# B&R Automation Studio project RTFProj (part 5)

#### test.c - Init, cyclic, exit code
```c
/*********************************************************************************************
* B&R Automation - Perfection in Automation (https://www.br-automation.com)
    ******************************************************************************************
    * Program 	    : Master's Thesis - Soccer Table (Table Football - real game)
    * Author  	    : Roman Parak
    * Created 	    : date ...
	* University    : Brno University of Technology(BUT)
	* Faculty       : Faculty of Mechanical Engineering(FME)
	* Study Program : Applied Computer Science and Control
	* Institute     : Institute of Automation and Computer Science
**********************************************************************************************
* Implementation OF PROGRAM Test(Real_Game/Technology/Test/Program/test.h)
**********************************************************************************************/

/*************************** LIBRARIES *********************************/
#include <bur/plc.h>
#include <bur/plctypes.h>
#include <stdio.h>
#include <math.h>

#include "rp_funcx1.h"
#include "Structures/test_str.h"
#include "Functions/test_fce.h"

#ifdef _DEFAULT_INCLUDES
	#include <AsDefault.h>
#endif

/*************************** DEFINITIONS *******************************/
#define EACH_FORMATION 1;

/************************ LOCAL VARIABLES ******************************/
// struct - MpAlarmX
_LOCAL MpAlarmXListUIConnectType AlarmListUI_ConnectType;
_LOCAL MpAlarmXHistoryUIConnectType AlarmHistoryUI_ConnectType;
// udint
_LOCAL UDINT alarm_device_address;
// bool
_LOCAL BOOL start;
_LOCAL BOOL stop;
// usint
_LOCAL USINT max_numberOfFormation;
_LOCAL USINT i_axisNum;
// lreal
_LOCAL LREAL temp_lin;
_LOCAL LREAL temp_rot;
_LOCAL LREAL define_posRotary;
_LOCAL LREAL angle_ofRotation;
// state machine
_LOCAL rp_MainSteps soccer_step;

/**********************************************************************************************************/
/********************************************** INIT PROGRAM **********************************************/
/**********************************************************************************************************/
void _INIT ProgramInit(void)
{
    /*********************************** Declaration variables **********************************/
    // generally
    max_numberOfFormation = EACH_FORMATION;

    // axis type -> MAPP -> Name Mapp axes for testing
    // linear
    //gLinkAxes_linear[0] = gk_mappAxisL;
    /*
    gLinkAxes_linear[1] = df_mappAxisL;
    gLinkAxes_linear[2] = md_mappAxisL;
    gLinkAxes_linear[3] = fw_mappAxisL;
    */
    // rotary
    //gLinkAxes_rotary[0] = gk_mappAxisR;
   	/*
    gLinkAxes_rotary[1] = df_mappAxisR;
    gLinkAxes_rotary[2] = md_mappAxisR;
    gLinkAxes_rotary[3] = fw_mappAxisR;
    */
    /************************************ Control of AlarmX ************************************/

    // adjustment device name
    alarm_device_address = (UDINT) strcpy(mp_alarmX.deviceName_no1_exp,"EXPORT_HISTORY");
    // MpAlarmX Core
    mp_alarmX.mp_core.MpLink         = &gAlarmXCore;
    mp_alarmX.mp_core.Enable         = 1;
    // MpAlarmX ListUI
    mp_alarmX.mp_listUI.MpLink       = &gAlarmXCore;
    mp_alarmX.mp_listUI.Enable       = 1;
    mp_alarmX.mp_listUI.UIConnect    = &AlarmListUI_ConnectType;
    // MpAlarmX History
    mp_alarmX.mp_history.MpLink      = &gAlarmXHistory;
    mp_alarmX.mp_history.Enable      = 1;
    mp_alarmX.mp_history.DeviceName  = &mp_alarmX.deviceName_no1_exp;
    // MpAlarmX HistoryUI
    mp_alarmX.mp_historyUI.MpLink    = &gAlarmXHistory;
    mp_alarmX.mp_historyUI.Enable    = 1;
    mp_alarmX.mp_historyUI.UIConnect = &AlarmHistoryUI_ConnectType;

    /************************************* Control of Axes **************************************/

    for(i_axisNum = 0; i_axisNum <= max_numberOfFormation - 1; i_axisNum++){
        // initialization ACOPOS variables through function(get_axisParam), that returns two variables type of UDINT
        // into the structure -> axesAcopos(have two parameters : linear, rotary)
        axis_acopos = get_axisParam(i_axisNum);
        // linear -> LinMot
        // linear axis basic
        mp_Axis.mp_axisLinear[i_axisNum].Enable     = 1;
        mp_Axis.mp_axisLinear[i_axisNum].MpLink     = &gLinkAxes_linear[i_axisNum];
        mp_Axis.mp_axisLinear[i_axisNum].Parameters = &mp_Axis.param_axisLinear[i_axisNum];
        mp_Axis.mp_axisLinear[i_axisNum].Axis       = axis_acopos.linear;
		// initialization parameters -> linear
		mp_Axis.param_axisLinear[i_axisNum].Home.Mode 	 		 	     = mpAXIS_HOME_MODE_BLOCK_TORQUE;
		mp_Axis.param_axisLinear[i_axisNum].Home.Position 		  	     = 900;
		mp_Axis.param_axisLinear[i_axisNum].Home.StartVelocity   		 = 350;
		mp_Axis.param_axisLinear[i_axisNum].Home.HomingVelocity  		 = 450;
		mp_Axis.param_axisLinear[i_axisNum].Home.Acceleration    		 = 350;
		mp_Axis.param_axisLinear[i_axisNum].Home.StartDirection  		 = mpAXIS_HOME_DIR_POSITIVE;
		mp_Axis.param_axisLinear[i_axisNum].Home.HomingDirection 		 = mpAXIS_HOME_DIR_NEGATIVE;
		mp_Axis.param_axisLinear[i_axisNum].Home.TorqueLimit	 		 = 0.05;
		mp_Axis.param_axisLinear[i_axisNum].Home.PositionErrorStopLimit	 = 900;
        // linear cyclic set
        mp_Axis.mp_cyclicSetLinear[i_axisNum].Enable     = 1;
        mp_Axis.mp_cyclicSetLinear[i_axisNum].MpLink     = &gLinkAxes_linear[i_axisNum];
        mp_Axis.mp_cyclicSetLinear[i_axisNum].Parameters = &mp_Axis.param_cyclicSetLinear[i_axisNum];
		// config
		mp_Axis.mp_configAxisLinear[i_axisNum].Enable 		 = 1;
		mp_Axis.mp_configAxisLinear[i_axisNum].MpLink 		 = &gLinkAxes_linear[i_axisNum];
		mp_Axis.mp_configAxisLinear[i_axisNum].Configuration = &mp_Axis.param_configAxisLinear[i_axisNum];
        // rotary -> EnDat
        // rotary axis basic
        mp_Axis.mp_axisRotary[i_axisNum].Enable     = 1;
        mp_Axis.mp_axisRotary[i_axisNum].MpLink     = &gLinkAxes_rotary[i_axisNum];
        mp_Axis.mp_axisRotary[i_axisNum].Parameters = &mp_Axis.param_axisRotary[i_axisNum];
        mp_Axis.mp_axisRotary[i_axisNum].Axis       = axis_acopos.rotary;
        // rotary cyclic set
        mp_Axis.mp_cyclicSetRotary[i_axisNum].Enable     = 1;
        mp_Axis.mp_cyclicSetRotary[i_axisNum].MpLink     = &gLinkAxes_rotary[i_axisNum];
        mp_Axis.mp_cyclicSetRotary[i_axisNum].Parameters = &mp_Axis.param_cyclicSetRotary[i_axisNum];
		// config
		mp_Axis.mp_configAxisRotary[i_axisNum].Enable 		 = 1;
		mp_Axis.mp_configAxisRotary[i_axisNum].MpLink 		 = &gLinkAxes_rotary[i_axisNum];
		mp_Axis.mp_configAxisRotary[i_axisNum].Configuration = &mp_Axis.param_configAxisRotary[i_axisNum];
		// temperature - linear
		mp_Axis.param_axisLinear[i_axisNum].CyclicRead.MotorTempMode = mpAXIS_READ_POLLING_1s;
		// temperature - rotary
		mp_Axis.param_axisRotary[i_axisNum].CyclicRead.MotorTempMode = mpAXIS_READ_POLLING_1s;
    }
	// initializatiom temp
	temp_lin = 0;
	temp_rot = 0;
	define_posRotary = 118520697;
	angle_ofRotation = 0;
	// initialization state machine
	soccer_step = STEP_INITIALIZATION;
}

/**********************************************************************************************************/
/********************************************** MAIN PROGRAM **********************************************/
/**********************************************************************************************************/
void _CYCLIC ProgramCyclic(void)
{
	// initializatiom temp
	temp_lin = mp_Axis.mp_axisLinear[0].Info.CyclicRead.MotorTemperature.Value;
	temp_rot = mp_Axis.mp_axisRotary[0].Info.CyclicRead.MotorTemperature.Value;

	switch(soccer_step)
	{
		case STEP_INITIALIZATION:
			{
				if(mp_Axis.mp_axisLinear[0].Active == 1 && mp_Axis.mp_axisRotary[0].Active == 1){
					angle_ofRotation = get_rotationalPostition(mp_Axis.mp_axisRotary[0].Position,define_posRotary);

					if(labs(angle_ofRotation) <= 3600){
						mp_Axis.param_axisRotary[0].Home.Position = angle_ofRotation;
						soccer_step = STEP_INITIALIZATION0;
					}
				}
			}
			break;
		case STEP_INITIALIZATION0:
			{
				if(mp_Axis.mp_axisLinear[0].Error == 1 && mp_Axis.mp_axisRotary[0].Error == 0){
					soccer_step = STEP_ERROR1;
				}else if(mp_Axis.mp_axisLinear[0].StatusID < 0 || mp_Axis.mp_axisRotary[0].StatusID < 0){
					soccer_step = STEP_ERROR2;
				}else {
					if(mp_Axis.mp_axisLinear[0].IsHomed == 1 && mp_Axis.mp_axisRotary[0].IsHomed == 1){
						soccer_step = STEP_RUN7;
					}else{
						soccer_step = STEP_INITIALIZATION1;
					}
				}
			}
			break;
		case STEP_INITIALIZATION1:
			{
				if(start == 1){
					mp_Axis.mp_axisLinear[0].Power = 1;
					mp_Axis.mp_axisRotary[0].Power = 1;

					if(mp_alarmX.mp_core.ActiveAlarms == 1){
						soccer_step = STEP_ERROR1;
					}else if(stop == 1){
						soccer_step = STEP_STOP1;
					}else{
						if(mp_Axis.mp_axisLinear[0].PowerOn == 1 && mp_Axis.mp_axisRotary[0].PowerOn == 1){
							soccer_step = STEP_INITIALIZATION2;
						}
					}
				}
			}
			break;
		case STEP_INITIALIZATION2:
			{
				mp_Axis.mp_axisLinear[0].Update = 1;
				mp_Axis.mp_axisRotary[0].Update = 1;

				if(mp_alarmX.mp_core.ActiveAlarms == 1){
					soccer_step = STEP_ERROR1;
				}else if(stop == 1){
					soccer_step = STEP_STOP1;
				}else{
					if(mp_Axis.mp_axisLinear[0].UpdateDone == 1 && mp_Axis.mp_axisRotary[0].UpdateDone == 1){
						mp_Axis.mp_axisLinear[0].Update = 0;
						mp_Axis.mp_axisRotary[0].Update = 0;
						soccer_step = STEP_INITIALIZATION3;
					}
				}
			}
			break;
		case STEP_INITIALIZATION3:
			{
				mp_Axis.mp_axisRotary[0].Home = 1;

				if(mp_alarmX.mp_core.ActiveAlarms == 1){
					soccer_step = STEP_ERROR1;
				}else if(stop == 1){
					soccer_step = STEP_STOP1;
				}else{
					if(mp_Axis.mp_axisRotary[0].IsHomed == 1){
						mp_Axis.mp_axisRotary[0].Home = 0;
						soccer_step = STEP_INITIALIZATION4;
					}
				}
			}
			break;
		case STEP_INITIALIZATION4:
			{
				mp_Axis.param_cyclicSetRotary[0].Acceleration = 2000;
				mp_Axis.param_cyclicSetRotary[0].Deceleration = 2000;
				mp_Axis.param_cyclicSetRotary[0].PositionModeMaxVelocity = 85000;
				mp_Axis.mp_cyclicSetRotary[0].Velocity 	 = 1000;
				mp_Axis.mp_cyclicSetRotary[0].Position	 = 0;

				mp_Axis.mp_cyclicSetRotary[0].Update = 1;
				if(mp_alarmX.mp_core.ActiveAlarms == 1){
					soccer_step = STEP_ERROR1;
				}else if(stop == 1){
					soccer_step = STEP_STOP1;
				}else{
					if(mp_Axis.mp_cyclicSetRotary[0].UpdateDone == 1){
						mp_Axis.mp_cyclicSetRotary[0].Update = 0;
						if(mp_Axis.mp_cyclicSetRotary[0].CommandBusy == 0 && mp_Axis.mp_cyclicSetRotary[0].CyclicSetActive == 0){
							soccer_step = STEP_INITIALIZATION5;
						}
					}
				}
			}
			break;
		case STEP_INITIALIZATION5:
			{
				mp_Axis.mp_cyclicSetRotary[0].CyclicPosition = 1;
				if(mp_alarmX.mp_core.ActiveAlarms == 1){
					soccer_step = STEP_ERROR1;
				}else if(stop == 1){
					soccer_step = STEP_STOP1;
				}else{
					if(mp_Axis.mp_cyclicSetRotary[0].Info.SlavePosition == 0){
						mp_Axis.mp_cyclicSetRotary[0].CyclicPosition = 0;
						if(mp_Axis.mp_cyclicSetRotary[0].CommandBusy == 0 && mp_Axis.mp_cyclicSetRotary[0].CyclicSetActive == 0){
							soccer_step = STEP_INITIALIZATION6;
						}
					}
				}
			}
			break;
		case STEP_INITIALIZATION6:
			{
				mp_Axis.mp_axisLinear[0].Home = 1;

				if(mp_alarmX.mp_core.ActiveAlarms == 1){
					soccer_step = STEP_ERROR1;
				}else if(stop == 1){
					soccer_step = STEP_STOP1;
				}else{
					if(mp_Axis.mp_axisLinear[0].IsHomed == 1){
						mp_Axis.mp_axisLinear[0].Home = 0;
						soccer_step = STEP_START;
					}
				}
			}
			break;
		case STEP_START:
			{
				mp_Axis.param_cyclicSetLinear[0].Acceleration = 400000;
				mp_Axis.param_cyclicSetLinear[0].Deceleration = 400000;
				mp_Axis.param_cyclicSetLinear[0].PositionModeMaxVelocity = 30000;
				mp_Axis.mp_cyclicSetLinear[0].Velocity = 19000;
				mp_Axis.mp_cyclicSetLinear[0].Position = 0;

				mp_Axis.mp_cyclicSetLinear[0].Update = 1;
				if(mp_alarmX.mp_core.ActiveAlarms == 1){
					soccer_step = STEP_ERROR1;
				}else if(stop == 1){
					soccer_step = STEP_STOP1;
				}else{
					if(mp_Axis.mp_cyclicSetLinear[0].UpdateDone == 1){
						mp_Axis.mp_cyclicSetLinear[0].Update = 0;
						if(mp_Axis.mp_cyclicSetLinear[0].CommandBusy == 0 && mp_Axis.mp_cyclicSetLinear[0].CyclicSetActive == 0){
							soccer_step = STEP_RUN1;
						}
					}
				}
			}
			break;
		case STEP_RUN1:
			{
				mp_Axis.mp_cyclicSetLinear[0].CyclicPosition = 1;
				if(mp_alarmX.mp_core.ActiveAlarms == 1){
					soccer_step = STEP_ERROR1;
				}else if(stop == 1){
					soccer_step = STEP_STOP1;
				}else{
					if(mp_Axis.mp_cyclicSetLinear[0].Info.SlavePosition == 0){
						mp_Axis.mp_cyclicSetLinear[0].CyclicPosition = 0;
						if(mp_Axis.mp_cyclicSetLinear[0].CommandBusy == 0 && mp_Axis.mp_cyclicSetLinear[0].CyclicSetActive == 0){
							soccer_step = STEP_RUN2;
						}
					}
				}
			}
			break;
		case STEP_RUN2:
			{
				mp_Axis.param_cyclicSetRotary[0].Acceleration = 125000;
				mp_Axis.param_cyclicSetRotary[0].Deceleration = 125000;
				mp_Axis.param_cyclicSetRotary[0].PositionModeMaxVelocity = 85000;
				mp_Axis.mp_cyclicSetRotary[0].Velocity 	 = 10000;
				mp_Axis.mp_cyclicSetRotary[0].Position	 = -800;

				mp_Axis.mp_cyclicSetRotary[0].Update = 1;
				if(mp_alarmX.mp_core.ActiveAlarms == 1){
					soccer_step = STEP_ERROR1;
				}else if(stop == 1){
					soccer_step = STEP_STOP1;
				}else{
					if(mp_Axis.mp_cyclicSetRotary[0].UpdateDone == 1){
						mp_Axis.mp_cyclicSetRotary[0].Update = 0;
						if(mp_Axis.mp_cyclicSetRotary[0].CommandBusy == 0 && mp_Axis.mp_cyclicSetRotary[0].CyclicSetActive == 0){
							soccer_step = STEP_RUN3;
						}
					}
				}
			}
			break;
		case STEP_RUN3:
			{
				mp_Axis.mp_cyclicSetRotary[0].CyclicPosition = 1;
				if(mp_alarmX.mp_core.ActiveAlarms == 1){
					soccer_step = STEP_ERROR1;
				}else if(stop == 1){
					soccer_step = STEP_STOP1;
				}else{
					if(mp_Axis.mp_cyclicSetRotary[0].Info.SlavePosition == -800){
						mp_Axis.mp_cyclicSetRotary[0].CyclicPosition = 0;
						if(mp_Axis.mp_cyclicSetRotary[0].CommandBusy == 0 && mp_Axis.mp_cyclicSetRotary[0].CyclicSetActive == 0){
							soccer_step = STEP_RUN4;
						}
					}
				}
			}
			break;
		case STEP_RUN4:
			{
				mp_Axis.param_cyclicSetRotary[0].Acceleration = 125000;
				mp_Axis.param_cyclicSetRotary[0].Deceleration = 125000;
				mp_Axis.param_cyclicSetRotary[0].PositionModeMaxVelocity = 85000;
				mp_Axis.mp_cyclicSetRotary[0].Velocity 	 = 10000;
				mp_Axis.mp_cyclicSetRotary[0].Position	 = 800;

				mp_Axis.mp_cyclicSetRotary[0].Update = 1;
				if(mp_alarmX.mp_core.ActiveAlarms == 1){
					soccer_step = STEP_ERROR1;
				}else if(stop == 1){
					soccer_step = STEP_STOP1;
				}else{
					if(mp_Axis.mp_cyclicSetRotary[0].UpdateDone == 1){
						mp_Axis.mp_cyclicSetRotary[0].Update = 0;
						if(mp_Axis.mp_cyclicSetRotary[0].CommandBusy == 0 && mp_Axis.mp_cyclicSetRotary[0].CyclicSetActive == 0){
							soccer_step = STEP_RUN5;
						}
					}
				}
			}
			break;
		case STEP_RUN5:
			{
				mp_Axis.mp_cyclicSetRotary[0].CyclicPosition = 1;
				if(mp_alarmX.mp_core.ActiveAlarms == 1){
					soccer_step = STEP_ERROR1;
				}else if(stop == 1){
					soccer_step = STEP_STOP1;
				}else{
					if(mp_Axis.mp_cyclicSetRotary[0].Info.SlavePosition == 800){
						mp_Axis.mp_cyclicSetRotary[0].CyclicPosition = 0;
						if(mp_Axis.mp_cyclicSetRotary[0].CommandBusy == 0 && mp_Axis.mp_cyclicSetRotary[0].CyclicSetActive == 0){
							soccer_step = STEP_RUN6;
						}
					}
				}
			}
			break;
		case STEP_RUN6:
			{
				/*======================= END HOME =======================*/
				mp_Axis.param_cyclicSetRotary[0].Acceleration = 125000;
				mp_Axis.param_cyclicSetRotary[0].Deceleration = 125000;
				mp_Axis.param_cyclicSetRotary[0].PositionModeMaxVelocity = 85000;
				mp_Axis.mp_cyclicSetRotary[0].Velocity 	 = 10000;
				mp_Axis.mp_cyclicSetRotary[0].Position	 = 0;

				mp_Axis.mp_cyclicSetRotary[0].Update = 1;
				if(mp_alarmX.mp_core.ActiveAlarms == 1){
					soccer_step = STEP_ERROR1;
				}else if(stop == 1){
					soccer_step = STEP_STOP1;
				}else{
					if(mp_Axis.mp_cyclicSetRotary[0].UpdateDone == 1){
						mp_Axis.mp_cyclicSetRotary[0].Update = 0;
						if(mp_Axis.mp_cyclicSetRotary[0].CommandBusy == 0 && mp_Axis.mp_cyclicSetRotary[0].CyclicSetActive == 0){
							soccer_step = STEP_RUN7;
						}
					}
				}
			}
			break;
		case STEP_RUN7:
			{
				/*======================= START CYCLE =======================*/
				mp_Axis.mp_cyclicSetRotary[0].CyclicPosition = 1;
				if(mp_alarmX.mp_core.ActiveAlarms == 1){
					soccer_step = STEP_ERROR1;
				}else if(stop == 1){
					soccer_step = STEP_STOP1;
				}else{
					if(mp_Axis.mp_cyclicSetRotary[0].Info.SlavePosition == 0){
						mp_Axis.mp_cyclicSetRotary[0].CyclicPosition = 0;
						if(mp_Axis.mp_cyclicSetRotary[0].CommandBusy == 0 && mp_Axis.mp_cyclicSetRotary[0].CyclicSetActive == 0){
							soccer_step = STEP_RUN8;
						}
					}
				}
			}
			break;
		case STEP_RUN8:
			{
				// 250000,20000
				mp_Axis.param_cyclicSetLinear[0].Acceleration = 125000;
				mp_Axis.param_cyclicSetLinear[0].Deceleration = 125000;
				mp_Axis.param_cyclicSetLinear[0].PositionModeMaxVelocity = 30000;
				mp_Axis.mp_cyclicSetLinear[0].Velocity = 10000;
				mp_Axis.mp_cyclicSetLinear[0].Position = -800;

				mp_Axis.mp_cyclicSetLinear[0].Update = 1;
				if(mp_alarmX.mp_core.ActiveAlarms == 1){
					soccer_step = STEP_ERROR1;
				}else if(stop == 1){
					soccer_step = STEP_STOP1;
				}else{
					if(mp_Axis.mp_cyclicSetLinear[0].UpdateDone == 1){
						mp_Axis.mp_cyclicSetLinear[0].Update = 0;
						if(mp_Axis.mp_cyclicSetLinear[0].CommandBusy == 0 && mp_Axis.mp_cyclicSetLinear[0].CyclicSetActive == 0){
							soccer_step = STEP_RUN9;
						}
					}
				}
			}
			break;
		case STEP_RUN9:
			{
				mp_Axis.mp_cyclicSetLinear[0].CyclicPosition = 1;
				if(mp_alarmX.mp_core.ActiveAlarms == 1){
					soccer_step = STEP_ERROR1;
				}else if(stop == 1){
					soccer_step = STEP_STOP1;
				}else{
					if(mp_Axis.mp_cyclicSetLinear[0].Info.SlavePosition == -800){
						mp_Axis.mp_cyclicSetLinear[0].CyclicPosition = 0;
						if(mp_Axis.mp_cyclicSetLinear[0].CommandBusy == 0 && mp_Axis.mp_cyclicSetLinear[0].CyclicSetActive == 0){
							soccer_step = STEP_RUN10; // STEP_RUN24
						}
					}
				}
			}
			break;
		case STEP_RUN10:
			{
				mp_Axis.param_cyclicSetRotary[0].Acceleration = 31250;
				mp_Axis.param_cyclicSetRotary[0].Deceleration = 31250;
				mp_Axis.param_cyclicSetRotary[0].PositionModeMaxVelocity = 85000;
				mp_Axis.mp_cyclicSetRotary[0].Velocity 	 = 5000;
				mp_Axis.mp_cyclicSetRotary[0].Position	 = -800;

				mp_Axis.mp_cyclicSetRotary[0].Update = 1;
				if(mp_alarmX.mp_core.ActiveAlarms == 1){
					soccer_step = STEP_ERROR1;
				}else if(stop == 1){
					soccer_step = STEP_STOP1;
				}else{
					if(mp_Axis.mp_cyclicSetRotary[0].UpdateDone == 1){
						mp_Axis.mp_cyclicSetRotary[0].Update = 0;
						if(mp_Axis.mp_cyclicSetRotary[0].CommandBusy == 0 && mp_Axis.mp_cyclicSetRotary[0].CyclicSetActive == 0){
							soccer_step = STEP_RUN11;
						}
					}
				}
			}
			break;
		case STEP_RUN11:
			{
				mp_Axis.mp_cyclicSetRotary[0].CyclicPosition = 1;
				if(mp_alarmX.mp_core.ActiveAlarms == 1){
					soccer_step = STEP_ERROR1;
				}else if(stop == 1){
					soccer_step = STEP_STOP1;
				}else{
					if(mp_Axis.mp_cyclicSetRotary[0].Info.SlavePosition == -800){
						mp_Axis.mp_cyclicSetRotary[0].CyclicPosition = 0;
						if(mp_Axis.mp_cyclicSetRotary[0].CommandBusy == 0 && mp_Axis.mp_cyclicSetRotary[0].CyclicSetActive == 0){
							soccer_step = STEP_RUN12;
						}
					}
				}
			}
			break;
		case STEP_RUN12:
			{
				mp_Axis.param_cyclicSetRotary[0].Acceleration = 31250;
				mp_Axis.param_cyclicSetRotary[0].Deceleration = 31250;
				mp_Axis.param_cyclicSetRotary[0].PositionModeMaxVelocity = 85000;
				mp_Axis.mp_cyclicSetRotary[0].Velocity 	 = 5000;
				mp_Axis.mp_cyclicSetRotary[0].Position	 = 800;

				mp_Axis.mp_cyclicSetRotary[0].Update = 1;
				if(mp_alarmX.mp_core.ActiveAlarms == 1){
					soccer_step = STEP_ERROR1;
				}else if(stop == 1){
					soccer_step = STEP_STOP1;
				}else{
					if(mp_Axis.mp_cyclicSetRotary[0].UpdateDone == 1){
						mp_Axis.mp_cyclicSetRotary[0].Update = 0;
						if(mp_Axis.mp_cyclicSetRotary[0].CommandBusy == 0 && mp_Axis.mp_cyclicSetRotary[0].CyclicSetActive == 0){
							soccer_step = STEP_RUN13;
						}
					}
				}
			}
			break;
		case STEP_RUN13:
			{
				mp_Axis.mp_cyclicSetRotary[0].CyclicPosition = 1;
				if(mp_alarmX.mp_core.ActiveAlarms == 1){
					soccer_step = STEP_ERROR1;
				}else if(stop == 1){
					soccer_step = STEP_STOP1;
				}else{
					if(mp_Axis.mp_cyclicSetRotary[0].Info.SlavePosition == 800){
						mp_Axis.mp_cyclicSetRotary[0].CyclicPosition = 0;
						if(mp_Axis.mp_cyclicSetRotary[0].CommandBusy == 0 && mp_Axis.mp_cyclicSetRotary[0].CyclicSetActive == 0){
							soccer_step = STEP_RUN14;
						}
					}
				}
			}
			break;
		case STEP_RUN14:
			{
				mp_Axis.param_cyclicSetRotary[0].Acceleration = 31250;
				mp_Axis.param_cyclicSetRotary[0].Deceleration = 31250;
				mp_Axis.param_cyclicSetRotary[0].PositionModeMaxVelocity = 85000;
				mp_Axis.mp_cyclicSetRotary[0].Velocity 	 = 5000;
				mp_Axis.mp_cyclicSetRotary[0].Position	 = 0;

				mp_Axis.mp_cyclicSetRotary[0].Update = 1;
				if(mp_alarmX.mp_core.ActiveAlarms == 1){
					soccer_step = STEP_ERROR1;
				}else if(stop == 1){
					soccer_step = STEP_STOP1;
				}else{
					if(mp_Axis.mp_cyclicSetRotary[0].UpdateDone == 1){
						mp_Axis.mp_cyclicSetRotary[0].Update = 0;
						if(mp_Axis.mp_cyclicSetRotary[0].CommandBusy == 0 && mp_Axis.mp_cyclicSetRotary[0].CyclicSetActive == 0){
							soccer_step = STEP_RUN15;
						}
					}
				}
			}
			break;
		case STEP_RUN15:
			{
				mp_Axis.mp_cyclicSetRotary[0].CyclicPosition = 1;
				if(mp_alarmX.mp_core.ActiveAlarms == 1){
					soccer_step = STEP_ERROR1;
				}else if(stop == 1){
					soccer_step = STEP_STOP1;
				}else{
					if(mp_Axis.mp_cyclicSetRotary[0].Info.SlavePosition == 0){
						mp_Axis.mp_cyclicSetRotary[0].CyclicPosition = 0;
						if(mp_Axis.mp_cyclicSetRotary[0].CommandBusy == 0 && mp_Axis.mp_cyclicSetRotary[0].CyclicSetActive == 0){
							soccer_step = STEP_RUN16; // STEP_RUN24
						}
					}
				}
			}
			break;
		case STEP_RUN16:
			{
				mp_Axis.param_cyclicSetLinear[0].Acceleration = 600;
				mp_Axis.param_cyclicSetLinear[0].Deceleration = 600;
				mp_Axis.param_cyclicSetLinear[0].PositionModeMaxVelocity = 30000;
				mp_Axis.mp_cyclicSetLinear[0].Velocity = 2500;
				mp_Axis.mp_cyclicSetLinear[0].Position = 0;

				mp_Axis.mp_cyclicSetLinear[0].Update = 1;
				if(mp_alarmX.mp_core.ActiveAlarms == 1){
					soccer_step = STEP_ERROR1;
				}else if(stop == 1){
					soccer_step = STEP_STOP1;
				}else{
					if(mp_Axis.mp_cyclicSetLinear[0].UpdateDone == 1){
						mp_Axis.mp_cyclicSetLinear[0].Update = 0;
						if(mp_Axis.mp_cyclicSetLinear[0].CommandBusy == 0 && mp_Axis.mp_cyclicSetLinear[0].CyclicSetActive == 0){
							soccer_step = STEP_RUN17;
						}
					}
				}
			}
			break;
		case STEP_RUN17:
			{
				mp_Axis.mp_cyclicSetLinear[0].CyclicPosition = 1;
				if(mp_alarmX.mp_core.ActiveAlarms == 1){
					soccer_step = STEP_ERROR1;
				}else if(stop == 1){
					soccer_step = STEP_STOP1;
				}else{
					if(mp_Axis.mp_cyclicSetLinear[0].Info.SlavePosition == 0){
						mp_Axis.mp_cyclicSetLinear[0].CyclicPosition = 0;
						if(mp_Axis.mp_cyclicSetLinear[0].CommandBusy == 0 && mp_Axis.mp_cyclicSetLinear[0].CyclicSetActive == 0){
							soccer_step = STEP_RUN18;
						}
					}
				}
			}
			break;
		case STEP_RUN18:
			{
				mp_Axis.param_cyclicSetRotary[0].Acceleration = 3900000;
				mp_Axis.param_cyclicSetRotary[0].Deceleration = 3900000;
				mp_Axis.param_cyclicSetRotary[0].PositionModeMaxVelocity = 85000;
				mp_Axis.mp_cyclicSetRotary[0].Velocity 	 = 84000;
				mp_Axis.mp_cyclicSetRotary[0].Position	 = -800;

				mp_Axis.mp_cyclicSetRotary[0].Update = 1;
				if(mp_alarmX.mp_core.ActiveAlarms == 1){
					soccer_step = STEP_ERROR1;
				}else if(stop == 1){
					soccer_step = STEP_STOP1;
				}else{
					if(mp_Axis.mp_cyclicSetRotary[0].UpdateDone == 1){
						mp_Axis.mp_cyclicSetRotary[0].Update = 0;
						if(mp_Axis.mp_cyclicSetRotary[0].CommandBusy == 0 && mp_Axis.mp_cyclicSetRotary[0].CyclicSetActive == 0){
							soccer_step = STEP_RUN19;
						}
					}
				}
			}
			break;
		case STEP_RUN19:
			{
				mp_Axis.mp_cyclicSetRotary[0].CyclicPosition = 1;
				if(mp_alarmX.mp_core.ActiveAlarms == 1){
					soccer_step = STEP_ERROR1;
				}else if(stop == 1){
					soccer_step = STEP_STOP1;
				}else{
					if(mp_Axis.mp_cyclicSetRotary[0].Info.SlavePosition == -800){
						mp_Axis.mp_cyclicSetRotary[0].CyclicPosition = 0;
						if(mp_Axis.mp_cyclicSetRotary[0].CommandBusy == 0 && mp_Axis.mp_cyclicSetRotary[0].CyclicSetActive == 0){
							soccer_step = STEP_RUN20;
						}
					}
				}
			}
			break;
		case STEP_RUN20:
			{
				mp_Axis.param_cyclicSetRotary[0].Acceleration = 3900000;
				mp_Axis.param_cyclicSetRotary[0].Deceleration = 3900000;
				mp_Axis.param_cyclicSetRotary[0].PositionModeMaxVelocity = 85000;
				mp_Axis.mp_cyclicSetRotary[0].Velocity 	 = 80000;
				mp_Axis.mp_cyclicSetRotary[0].Position	 = 800;

				mp_Axis.mp_cyclicSetRotary[0].Update = 1;
				if(mp_alarmX.mp_core.ActiveAlarms == 1){
					soccer_step = STEP_ERROR1;
				}else if(stop == 1){
					soccer_step = STEP_STOP1;
				}else{
					if(mp_Axis.mp_cyclicSetRotary[0].UpdateDone == 1){
						mp_Axis.mp_cyclicSetRotary[0].Update = 0;
						if(mp_Axis.mp_cyclicSetRotary[0].CommandBusy == 0 && mp_Axis.mp_cyclicSetRotary[0].CyclicSetActive == 0){
							soccer_step = STEP_RUN21;
						}
					}
				}
			}
			break;
		case STEP_RUN21:
			{
				mp_Axis.mp_cyclicSetRotary[0].CyclicPosition = 1;
				if(mp_alarmX.mp_core.ActiveAlarms == 1){
					soccer_step = STEP_ERROR1;
				}else if(stop == 1){
					soccer_step = STEP_STOP1;
				}else{
					if(mp_Axis.mp_cyclicSetRotary[0].Info.SlavePosition == 800){
						mp_Axis.mp_cyclicSetRotary[0].CyclicPosition = 0;
						if(mp_Axis.mp_cyclicSetRotary[0].CommandBusy == 0 && mp_Axis.mp_cyclicSetRotary[0].CyclicSetActive == 0){
							soccer_step = STEP_RUN22;
						}
					}
				}
			}
			break;
		case STEP_RUN22:
			{
				mp_Axis.param_cyclicSetRotary[0].Acceleration = 3900000;
				mp_Axis.param_cyclicSetRotary[0].Deceleration = 3900000;
				mp_Axis.param_cyclicSetRotary[0].PositionModeMaxVelocity = 85000;
				mp_Axis.mp_cyclicSetRotary[0].Velocity 	 = 80000;
				mp_Axis.mp_cyclicSetRotary[0].Position	 = 0;

				mp_Axis.mp_cyclicSetRotary[0].Update = 1;
				if(mp_alarmX.mp_core.ActiveAlarms == 1){
					soccer_step = STEP_ERROR1;
				}else if(stop == 1){
					soccer_step = STEP_STOP1;
				}else{
					if(mp_Axis.mp_cyclicSetRotary[0].UpdateDone == 1){
						mp_Axis.mp_cyclicSetRotary[0].Update = 0;
						if(mp_Axis.mp_cyclicSetRotary[0].CommandBusy == 0 && mp_Axis.mp_cyclicSetRotary[0].CyclicSetActive == 0){
							soccer_step = STEP_RUN23;
						}
					}
				}
			}
			break;
		case STEP_RUN23:
			{
				mp_Axis.mp_cyclicSetRotary[0].CyclicPosition = 1;
				if(mp_alarmX.mp_core.ActiveAlarms == 1){
					soccer_step = STEP_ERROR1;
				}else if(stop == 1){
					soccer_step = STEP_STOP1;
				}else{
					if(mp_Axis.mp_cyclicSetRotary[0].Info.SlavePosition == 0){
						mp_Axis.mp_cyclicSetRotary[0].CyclicPosition = 0;
						if(mp_Axis.mp_cyclicSetRotary[0].CommandBusy == 0 && mp_Axis.mp_cyclicSetRotary[0].CyclicSetActive == 0){
							soccer_step = STEP_RUN24;
						}
					}
				}
			}
			break;
		case STEP_RUN24:
			{
				// 250000, 20000
				mp_Axis.param_cyclicSetLinear[0].Acceleration = 281250;
				mp_Axis.param_cyclicSetLinear[0].Deceleration = 281250;
				mp_Axis.param_cyclicSetLinear[0].PositionModeMaxVelocity = 30000;
				mp_Axis.mp_cyclicSetLinear[0].Velocity = 15000;
				mp_Axis.mp_cyclicSetLinear[0].Position = 800;

				mp_Axis.mp_cyclicSetLinear[0].Update = 1;
				if(mp_alarmX.mp_core.ActiveAlarms == 1){
					soccer_step = STEP_ERROR1;
				}else if(stop == 1){
					soccer_step = STEP_STOP1;
				}else{
					if(mp_Axis.mp_cyclicSetLinear[0].UpdateDone == 1){
						mp_Axis.mp_cyclicSetLinear[0].Update = 0;
						if(mp_Axis.mp_cyclicSetLinear[0].CommandBusy == 0 && mp_Axis.mp_cyclicSetLinear[0].CyclicSetActive == 0){
							soccer_step = STEP_RUN25;
						}
					}
				}
			}
			break;
		case STEP_RUN25:
			{
				mp_Axis.mp_cyclicSetLinear[0].CyclicPosition = 1;
				if(mp_alarmX.mp_core.ActiveAlarms == 1){
					soccer_step = STEP_ERROR1;
				}else if(stop == 1){
					soccer_step = STEP_STOP1;
				}else{
					if(mp_Axis.mp_cyclicSetLinear[0].Info.SlavePosition == 800){
						mp_Axis.mp_cyclicSetLinear[0].CyclicPosition = 0;
						if(mp_Axis.mp_cyclicSetLinear[0].CommandBusy == 0 && mp_Axis.mp_cyclicSetLinear[0].CyclicSetActive == 0){
							soccer_step = STEP_RUN26; // STEP_RUN8
						}
					}
				}
			}
			break;
		case STEP_RUN26:
			{
				mp_Axis.param_cyclicSetRotary[0].Acceleration = 3125000;
				mp_Axis.param_cyclicSetRotary[0].Deceleration = 3125000;
				mp_Axis.param_cyclicSetRotary[0].PositionModeMaxVelocity = 85000;
				mp_Axis.mp_cyclicSetRotary[0].Velocity 	 = 50000;
				mp_Axis.mp_cyclicSetRotary[0].Position	 = -800;

				mp_Axis.mp_cyclicSetRotary[0].Update = 1;
				if(mp_alarmX.mp_core.ActiveAlarms == 1){
					soccer_step = STEP_ERROR1;
				}else if(stop == 1){
					soccer_step = STEP_STOP1;
				}else{
					if(mp_Axis.mp_cyclicSetRotary[0].UpdateDone == 1){
						mp_Axis.mp_cyclicSetRotary[0].Update = 0;
						if(mp_Axis.mp_cyclicSetRotary[0].CommandBusy == 0 && mp_Axis.mp_cyclicSetRotary[0].CyclicSetActive == 0){
							soccer_step = STEP_RUN27;
						}
					}
				}
			}
			break;
		case STEP_RUN27:
			{
				mp_Axis.mp_cyclicSetRotary[0].CyclicPosition = 1;
				if(mp_alarmX.mp_core.ActiveAlarms == 1){
					soccer_step = STEP_ERROR1;
				}else if(stop == 1){
					soccer_step = STEP_STOP1;
				}else{
					if(mp_Axis.mp_cyclicSetRotary[0].Info.SlavePosition == -800){
						mp_Axis.mp_cyclicSetRotary[0].CyclicPosition = 0;
						if(mp_Axis.mp_cyclicSetRotary[0].CommandBusy == 0 && mp_Axis.mp_cyclicSetRotary[0].CyclicSetActive == 0){
							soccer_step = STEP_RUN28;
						}
					}
				}
			}
			break;
		case STEP_RUN28:
			{
				mp_Axis.param_cyclicSetRotary[0].Acceleration = 11300;
				mp_Axis.param_cyclicSetRotary[0].Deceleration = 11300;
				mp_Axis.param_cyclicSetRotary[0].PositionModeMaxVelocity = 85000;
				mp_Axis.mp_cyclicSetRotary[0].Velocity 	 = 3000;
				mp_Axis.mp_cyclicSetRotary[0].Position	 = 800;

				mp_Axis.mp_cyclicSetRotary[0].Update = 1;
				if(mp_alarmX.mp_core.ActiveAlarms == 1){
					soccer_step = STEP_ERROR1;
				}else if(stop == 1){
					soccer_step = STEP_STOP1;
				}else{
					if(mp_Axis.mp_cyclicSetRotary[0].UpdateDone == 1){
						mp_Axis.mp_cyclicSetRotary[0].Update = 0;
						if(mp_Axis.mp_cyclicSetRotary[0].CommandBusy == 0 && mp_Axis.mp_cyclicSetRotary[0].CyclicSetActive == 0){
							soccer_step = STEP_RUN29;
						}
					}
				}
			}
			break;
		case STEP_RUN29:
			{
				mp_Axis.mp_cyclicSetRotary[0].CyclicPosition = 1;
				if(mp_alarmX.mp_core.ActiveAlarms == 1){
					soccer_step = STEP_ERROR1;
				}else if(stop == 1){
					soccer_step = STEP_STOP1;
				}else{
					if(mp_Axis.mp_cyclicSetRotary[0].Info.SlavePosition == 800){
						mp_Axis.mp_cyclicSetRotary[0].CyclicPosition = 0;
						if(mp_Axis.mp_cyclicSetRotary[0].CommandBusy == 0 && mp_Axis.mp_cyclicSetRotary[0].CyclicSetActive == 0){
							soccer_step = STEP_RUN30;
						}
					}
				}
			}
			break;
		case STEP_RUN30:
			{
				mp_Axis.param_cyclicSetRotary[0].Acceleration = 1000;
				mp_Axis.param_cyclicSetRotary[0].Deceleration = 1000;
				mp_Axis.param_cyclicSetRotary[0].PositionModeMaxVelocity = 85000;
				mp_Axis.mp_cyclicSetRotary[0].Velocity 	 = 1000;
				mp_Axis.mp_cyclicSetRotary[0].Position	 = 0;

				mp_Axis.mp_cyclicSetRotary[0].Update = 1;
				if(mp_alarmX.mp_core.ActiveAlarms == 1){
					soccer_step = STEP_ERROR1;
				}else if(stop == 1){
					soccer_step = STEP_STOP1;
				}else{
					if(mp_Axis.mp_cyclicSetRotary[0].UpdateDone == 1){
						mp_Axis.mp_cyclicSetRotary[0].Update = 0;
						if(mp_Axis.mp_cyclicSetRotary[0].CommandBusy == 0 && mp_Axis.mp_cyclicSetRotary[0].CyclicSetActive == 0){
							soccer_step = STEP_RUN31;
						}
					}
				}
			}
			break;
		case STEP_RUN31:
			{
				mp_Axis.mp_cyclicSetRotary[0].CyclicPosition = 1;
				if(mp_alarmX.mp_core.ActiveAlarms == 1){
					soccer_step = STEP_ERROR1;
				}else if(stop == 1){
					soccer_step = STEP_STOP1;
				}else{
					if(mp_Axis.mp_cyclicSetRotary[0].Info.SlavePosition == 0){
						mp_Axis.mp_cyclicSetRotary[0].CyclicPosition = 0;
						if(mp_Axis.mp_cyclicSetRotary[0].CommandBusy == 0 && mp_Axis.mp_cyclicSetRotary[0].CyclicSetActive == 0){
							soccer_step = STEP_RUN32; //STEP_RUN8
						}
					}
				}
			}
			break;
		case STEP_RUN32:
			{
				mp_Axis.param_cyclicSetLinear[0].Acceleration = 440000;
				mp_Axis.param_cyclicSetLinear[0].Deceleration = 440000;
				mp_Axis.param_cyclicSetLinear[0].PositionModeMaxVelocity = 30000;
				mp_Axis.mp_cyclicSetLinear[0].Velocity = 20000;
				mp_Axis.mp_cyclicSetLinear[0].Position = 0;

				mp_Axis.mp_cyclicSetLinear[0].Update = 1;
				if(mp_alarmX.mp_core.ActiveAlarms == 1){
					soccer_step = STEP_ERROR1;
				}else if(stop == 1){
					soccer_step = STEP_STOP1;
				}else{
					if(mp_Axis.mp_cyclicSetLinear[0].UpdateDone == 1){
						mp_Axis.mp_cyclicSetLinear[0].Update = 0;
						if(mp_Axis.mp_cyclicSetLinear[0].CommandBusy == 0 && mp_Axis.mp_cyclicSetLinear[0].CyclicSetActive == 0){
							soccer_step = STEP_RUN33;
						}
					}
				}
			}
			break;
		case STEP_RUN33:
			{
				mp_Axis.mp_cyclicSetLinear[0].CyclicPosition = 1;
				if(mp_alarmX.mp_core.ActiveAlarms == 1){
					soccer_step = STEP_ERROR1;
				}else if(stop == 1){
					soccer_step = STEP_STOP1;
				}else{
					if(mp_Axis.mp_cyclicSetLinear[0].Info.SlavePosition == 0){
						mp_Axis.mp_cyclicSetLinear[0].CyclicPosition = 0;
						if(mp_Axis.mp_cyclicSetLinear[0].CommandBusy == 0 && mp_Axis.mp_cyclicSetLinear[0].CyclicSetActive == 0){
							soccer_step = STEP_RUN34;
						}
					}
				}
			}
			break;
		case STEP_RUN34:
			{
				mp_Axis.param_cyclicSetRotary[0].Acceleration = 3900000;
				mp_Axis.param_cyclicSetRotary[0].Deceleration = 3900000;
				mp_Axis.param_cyclicSetRotary[0].PositionModeMaxVelocity = 85000;
				mp_Axis.mp_cyclicSetRotary[0].Velocity 	 = 84000;
				mp_Axis.mp_cyclicSetRotary[0].Position	 = -800;

				mp_Axis.mp_cyclicSetRotary[0].Update = 1;
				if(mp_alarmX.mp_core.ActiveAlarms == 1){
					soccer_step = STEP_ERROR1;
				}else if(stop == 1){
					soccer_step = STEP_STOP1;
				}else{
					if(mp_Axis.mp_cyclicSetRotary[0].UpdateDone == 1){
						mp_Axis.mp_cyclicSetRotary[0].Update = 0;
						if(mp_Axis.mp_cyclicSetRotary[0].CommandBusy == 0 && mp_Axis.mp_cyclicSetRotary[0].CyclicSetActive == 0){
							soccer_step = STEP_RUN35;
						}
					}
				}
			}
			break;
		case STEP_RUN35:
			{
				mp_Axis.mp_cyclicSetRotary[0].CyclicPosition = 1;
				if(mp_alarmX.mp_core.ActiveAlarms == 1){
					soccer_step = STEP_ERROR1;
				}else if(stop == 1){
					soccer_step = STEP_STOP1;
				}else{
					if(mp_Axis.mp_cyclicSetRotary[0].Info.SlavePosition == -800){
						mp_Axis.mp_cyclicSetRotary[0].CyclicPosition = 0;
						if(mp_Axis.mp_cyclicSetRotary[0].CommandBusy == 0 && mp_Axis.mp_cyclicSetRotary[0].CyclicSetActive == 0){
							soccer_step = STEP_RUN36;
						}
					}
				}
			}
			break;
		case STEP_RUN36:
			{
				mp_Axis.param_cyclicSetRotary[0].Acceleration = 3900000;
				mp_Axis.param_cyclicSetRotary[0].Deceleration = 3900000;
				mp_Axis.param_cyclicSetRotary[0].PositionModeMaxVelocity = 85000;
				mp_Axis.mp_cyclicSetRotary[0].Velocity 	 = 84000;
				mp_Axis.mp_cyclicSetRotary[0].Position	 = 800;

				mp_Axis.mp_cyclicSetRotary[0].Update = 1;
				if(mp_alarmX.mp_core.ActiveAlarms == 1){
					soccer_step = STEP_ERROR1;
				}else if(stop == 1){
					soccer_step = STEP_STOP1;
				}else{
					if(mp_Axis.mp_cyclicSetRotary[0].UpdateDone == 1){
						mp_Axis.mp_cyclicSetRotary[0].Update = 0;
						if(mp_Axis.mp_cyclicSetRotary[0].CommandBusy == 0 && mp_Axis.mp_cyclicSetRotary[0].CyclicSetActive == 0){
							soccer_step = STEP_RUN37;
						}
					}
				}
			}
			break;
		case STEP_RUN37:
			{
				mp_Axis.mp_cyclicSetRotary[0].CyclicPosition = 1;
				if(mp_alarmX.mp_core.ActiveAlarms == 1){
					soccer_step = STEP_ERROR1;
				}else if(stop == 1){
					soccer_step = STEP_STOP1;
				}else{
					if(mp_Axis.mp_cyclicSetRotary[0].Info.SlavePosition == 800){
						mp_Axis.mp_cyclicSetRotary[0].CyclicPosition = 0;
						if(mp_Axis.mp_cyclicSetRotary[0].CommandBusy == 0 && mp_Axis.mp_cyclicSetRotary[0].CyclicSetActive == 0){
							soccer_step = STEP_RUN38;
						}
					}
				}
			}
			break;
		case STEP_RUN38:
			{
				mp_Axis.param_cyclicSetRotary[0].Acceleration = 61300;
				mp_Axis.param_cyclicSetRotary[0].Deceleration = 61300;
				mp_Axis.param_cyclicSetRotary[0].PositionModeMaxVelocity = 85000;
				mp_Axis.mp_cyclicSetRotary[0].Velocity 	 = 7000;
				mp_Axis.mp_cyclicSetRotary[0].Position	 = 0;

				mp_Axis.mp_cyclicSetRotary[0].Update = 1;
				if(mp_alarmX.mp_core.ActiveAlarms == 1){
					soccer_step = STEP_ERROR1;
				}else if(stop == 1){
					soccer_step = STEP_STOP1;
				}else{
					if(mp_Axis.mp_cyclicSetRotary[0].UpdateDone == 1){
						mp_Axis.mp_cyclicSetRotary[0].Update = 0;
						if(mp_Axis.mp_cyclicSetRotary[0].CommandBusy == 0 && mp_Axis.mp_cyclicSetRotary[0].CyclicSetActive == 0){
							soccer_step = STEP_RUN39;
						}
					}
				}
			}
			break;
		case STEP_RUN39:
			{
				mp_Axis.mp_cyclicSetRotary[0].CyclicPosition = 1;
				if(mp_alarmX.mp_core.ActiveAlarms == 1){
					soccer_step = STEP_ERROR1;
				}else if(stop == 1){
					soccer_step = STEP_STOP1;
				}else{
					if(mp_Axis.mp_cyclicSetRotary[0].Info.SlavePosition == 0){
						mp_Axis.mp_cyclicSetRotary[0].CyclicPosition = 0;
						if(mp_Axis.mp_cyclicSetRotary[0].CommandBusy == 0 && mp_Axis.mp_cyclicSetRotary[0].CyclicSetActive == 0){
							soccer_step = STEP_RUN8;
						}
					}
				}
			}
			break;
		case STEP_RUN40:
			{
				if(mp_alarmX.mp_core.ActiveAlarms == 1){
					soccer_step = STEP_ERROR1;
				}else if(stop == 1){
					soccer_step = STEP_STOP1;
				}else{
				}
			}
			break;
		case STEP_STOP1:
			{
				start = 0;
				mp_Axis.mp_axisLinear[0].Stop = 1;
				mp_Axis.mp_axisRotary[0].Stop = 1;

				if(mp_alarmX.mp_core.ActiveAlarms == 1){
					soccer_step = STEP_ERROR1;
				}else if(stop == 0){
					mp_Axis.mp_axisLinear[0].Stop = 0;
					mp_Axis.mp_axisRotary[0].Stop = 0;
					soccer_step = STEP_INITIALIZATION0;
				}
			}
			break;
		case STEP_ERROR1:
			{
				start = 0;
				stop  = 0;
				mp_Axis.mp_axisLinear[0].Stop = 0;
				mp_Axis.mp_axisRotary[0].Stop = 0;
				mp_Axis.mp_axisLinear[0].Power = 0;
				mp_Axis.mp_axisRotary[0].Power = 0;

				mp_Axis.mp_axisLinear[0].ErrorReset = 1;
				mp_Axis.mp_axisRotary[0].ErrorReset = 1;

				if(mp_Axis.mp_axisLinear[0].Error == 0 && mp_Axis.mp_axisRotary[0].Error == 0){
					mp_Axis.mp_axisLinear[0].ErrorReset = 0;
					mp_Axis.mp_axisRotary[0].ErrorReset = 0;

					soccer_step = STEP_INITIALIZATION0;
				}

			}
			break;
		case STEP_ERROR2:
			{
				mp_Axis.mp_axisLinear[0].ErrorReset = 1;
				mp_Axis.mp_axisRotary[0].ErrorReset = 1;

				if(mp_Axis.mp_axisLinear[0].StatusID >= 0 && mp_Axis.mp_axisRotary[0].StatusID >= 0){
					mp_Axis.mp_axisLinear[0].ErrorReset = 0;
					mp_Axis.mp_axisRotary[0].ErrorReset = 0;

					soccer_step = STEP_INITIALIZATION0;
				}
			}
			break;
	}

    /************************** Call function & function blocks **************************/
    // AlarmX
    MpAlarmXCore(&mp_alarmX.mp_core);
    MpAlarmXListUI(&mp_alarmX.mp_listUI);
    MpAlarmXHistory(&mp_alarmX.mp_history);
    MpAlarmXHistoryUI(&mp_alarmX.mp_historyUI);
    // Active AxisBasic & AxisCyclicSet -> through the individual functions
    start_axesBasic(max_numberOfFormation,&mp_Axis.mp_axisLinear,&mp_Axis.mp_axisRotary);
    start_axesCyclic(max_numberOfFormation,&mp_Axis.mp_cyclicSetLinear,&mp_Axis.mp_cyclicSetRotary);

}
```

#### test_str.h
```c
/*********************************************************************************************
* B&R Automation - Perfection in Automation (https://www.br-automation.com)
    ******************************************************************************************
    * Program 	    : Master's Thesis - Soccer Table (Table Football - real game)
    * Author  	    : Roman Parak
    * Created 	    : date ...
	* University    : Brno University of Technology(BUT)
	* Faculty       : Faculty of Mechanical Engineering(FME)
	* Study Program : Applied Computer Science and Control
	* Institute     : Institute of Automation and Computer Science
**********************************************************************************************
* Implementation OF PROGRAM Test(Real_Game/Technolog/Test/Structures/test_str.h)
**********************************************************************************************/

/*************************** LIBRARIES *********************************/
#include <bur/plc.h>
#include <bur/plctypes.h>
#include <AsString.h>
#include <AsWStr.h>

#ifdef _DEFAULT_INCLUDES
    #include <AsDefault.h>
#endif

/**********************************************************************************************************/
/************************************** STRUCTURE TYPE ****************************************************/
/**********************************************************************************************************/

/***************************** ALARM ***********************************/
typedef struct mappAlarmX_STR{
    // list
    struct MpAlarmXCore   mp_core;
    struct MpAlarmXListUI mp_listUI;
    // history
    struct    MpAlarmXHistory mp_history;
    struct    MpAlarmXHistoryUI mp_historyUI;
    plcstring deviceName_no1_exp[21];
} mappAlarmX_STR;

/***************************** AXIS ************************************/
typedef struct mappAxisBasic_STR{
    // === Linear Axes === //
    // axis basic
    struct MpAxisBasic        mp_axisLinear[4];
    struct MpAxisBasicParType param_axisLinear[4];
    // cyclic set
    struct MpAxisCyclicSet        mp_cyclicSetLinear[4];
    struct MpAxisCyclicSetParType param_cyclicSetLinear[4];
	// config
	struct MpAxisBasicConfig mp_configAxisLinear[4];
	struct MpAxisBasicConfigType param_configAxisLinear[4];
    // === Rotary Axes === //
    // axis basic
    struct MpAxisBasic        mp_axisRotary[4];
    struct MpAxisBasicParType param_axisRotary[4];
    // cyclic set
    struct MpAxisCyclicSet        mp_cyclicSetRotary[4];
    struct MpAxisCyclicSetParType param_cyclicSetRotary[4];
	// config
	struct MpAxisBasicConfig mp_configAxisRotary[4];
	struct MpAxisBasicConfigType param_configAxisRotary[4];
} mappAxisBasic_STR;

// auxiliary structures
typedef struct axesAcopos{
    UDINT linear;
    UDINT rotary;
}axesAcopos;

/**********************************************************************************************************/
/**************************************** GLOBAL VARIABLES ************************************************/
/**********************************************************************************************************/
// my structures
_GLOBAL mappAlarmX_STR mp_alarmX;
_GLOBAL mappAxisBasic_STR mp_Axis;
_GLOBAL axesAcopos axis_acopos;

// axis type -> ACOPOS
// goalkeeper
_GLOBAL ACP10AXIS_typ gkLinearW;
_GLOBAL ACP10AXIS_typ gkRotaryW;
// defender
/*
_GLOBAL ACP10AXIS_typ dfLinearX;
_GLOBAL ACP10AXIS_typ dfRotaryX;
// midfielder
_GLOBAL ACP10AXIS_typ mdLinearY;
_GLOBAL ACP10AXIS_typ mdRotaryY;
// forward
_GLOBAL ACP10AXIS_typ fwLinearZ;
_GLOBAL ACP10AXIS_typ fwRotaryZ;
*/
// axis type -> MAPP
_GLOBAL struct MpComIdentType gLinkAxes_rotary[4];
_GLOBAL struct MpComIdentType gLinkAxes_linear[4];

/**********************************************************************************************************/
/************************************** FUNCTIONS & FUNCTIONS BLOCKS **************************************/
/**********************************************************************************************************/
void start_axesBasic(USINT num_ofAxes,struct MpAxisBasic* axis_linear,struct MpAxisBasic* axis_rotary);
void start_axesCyclic(USINT num_ofAxes,struct MpAxisCyclicSet* cyclic_linear,struct MpAxisCyclicSet* cyclic_rotary);
struct axesAcopos get_axisParam(int idx_ofIteration);
```

#### test_fce.h
```c
/*********************************************************************************************
* B&R Automation - Perfection in Automation (https://www.br-automation.com)
    ******************************************************************************************
    * Program 	    : Master's Thesis - Soccer Table (Table Football - real game)
    * Author  	    : Roman Parak
    * Created 	    : date ...
	* University    : Brno University of Technology(BUT)
	* Faculty       : Faculty of Mechanical Engineering(FME)
	* Study Program : Applied Computer Science and Control
	* Institute     : Institute of Automation and Computer Science
**********************************************************************************************
* Implementation OF PROGRAM Test(Real_Game/Technolog/table_football/Functions/test_mapp_fce.h)
**********************************************************************************************/

/*************************** LIBRARIES *********************************/
#include <bur/plc.h>
#include <bur/plctypes.h>
#include <AsString.h>
#include <standard.h>
#include <AsWStr.h>
#include <stdio.h>
#include <math.h>

#ifdef _DEFAULT_INCLUDES
    #include <AsDefault.h>
#endif

/**********************************************************************************************************/
/************************************** FUNCTIONS & FUNCTIONS BLOCKS **************************************/
/**********************************************************************************************************/
void start_axesBasic(USINT num_ofAxes,struct MpAxisBasic* axis_linear,struct MpAxisBasic* axis_rotary){
    int i;
    // Axis Basic
    // function to start the individual axes
    // the cycle is carried out through number of axes
    for(i = 0; i <= num_ofAxes - 1; i++){
        // mapp axis basic
        MpAxisBasic(&axis_linear[i]);
        MpAxisBasic(&axis_rotary[i]);
    }
}

void start_axesCyclic(USINT num_ofAxes,struct MpAxisCyclicSet* cyclic_linear,struct MpAxisCyclicSet* cyclic_rotary){
    int i;
    // Axis Cyclic Set
    // function to start the individual axes
    // the cycle is carried out through number of axes
    for(i = 0; i <= num_ofAxes - 1; i++){
        // mapp axis cyclic set
        MpAxisCyclicSet(&cyclic_linear[i]);
        MpAxisCyclicSet(&cyclic_rotary[i]);
    }
}

struct axesAcopos get_axisParam(int idx_ofIteration){
    // input into the function is number of iteration(in the init part)
    // create auxiliary structures and enumeration type(for state machine)
    struct axesAcopos a;
    typedef enum {aNUM1 = 0, aNUM2, aNUM3, aNUM4}wState_ofAxes;
    wState_ofAxes new_idx; // initialize state machine
    new_idx = idx_ofIteration;
    // gradually into the state machine loading indexes from initialization part
    // and this run the function blocks
    // each state of machine has initialization both engines linear and rotary, on its own axis
    // output of this function is structure, that has two parameters(linear,rotary axis)
    switch(new_idx){
        case aNUM1:
			// Name real axes
			/*
            // goalkeeper
            a.linear = &gkLinearW;
            a.rotary = &gkRotaryW;
            return a;
            break;
        case aNUM2:
            // defender
            a.linear = &dfLinearX;
            a.rotary = &dfRotaryX;
            return a;
            break;
        case aNUM3:
            // midfielder
            a.linear = &mdLinearY;
            a.rotary = &mdRotaryY;
            return a;
            break;
        case aNUM4:
            // forward
            a.linear = &fwLinearZ;
            a.rotary = &fwRotaryZ;
            break;
        */
    }
}
```

### Program Logical/Real_Game/Technology/cam_sens_sd_s (ANSIC) - Lubo,Radek program for real game.

#### main_real.c - Init, cyclic, exit code
```c
/*********************************************************************************************
* B&R Automation - Perfection in Automation (https://www.br-automation.com)
    ******************************************************************************************
    * Program 	    : Bachelor's Thesis
    * Author  	    : Lubomir Bubenik, Radek Otradovský
    * Created 	    : date ...
	* University    : Brno University of Technology(BUT)
	* Faculty       : Faculty of Mechanical Engineering(FME), Faculty of Electrical Engineering and Communication(FEEC)
**********************************************************************************************
* Implementation OF PROGRAM cam_sens_sd_s(Real_Game/Technology/sim_cam_sens_sd_s/main_real.c)
**********************************************************************************************/

#include <bur/plctypes.h>
#include <AsMem.h>
#include <Camera.h>

#ifdef _DEFAULT_INCLUDES
#include <AsDefault.h>
#endif
#define Y_AXIS
#define ABS_F(X) ((X) < (0) ? -(X) : (X))
struct Buffer{
	REAL X;
	REAL Y;
	REAL TimeDiff;
};

_GLOBAL FBCamera_typ FBCamera_0;
_GLOBAL Light_typ Light_0;
_GLOBAL GoalKeeper_typ GoalKeeper_0;
_LOCAL struct Buffer BufferRes[20];
_LOCAL INT i;
_LOCAL INT tmp;
_LOCAL INT Reset;

void _INIT ProgramInit(void)
{
	FBCamera_0.Enable = 1;
	i = 0;
	tmp = 0;
	Reset = 0;
}

void _CYCLIC ProgramCyclic(void)
{

	FBCamera(&FBCamera_0);
	Light(&Light_0);
	GoalKeeper(&GoalKeeper_0);

	if ((FBCamera_0.isBallFound) || (tmp)){
		if (((ABS_F(FBCamera_0.Results.AxisX-FBCamera_0.Results.AxisXOld)) > 100) && (!tmp)){
			BufferRes[0].X = FBCamera_0.Results.AxisXOld;
			BufferRes[0].Y = FBCamera_0.Results.AxisYOld;
			BufferRes[0].TimeDiff = 0;

			BufferRes[1].X = FBCamera_0.Results.AxisX;
			BufferRes[1].Y = FBCamera_0.Results.AxisY;
			BufferRes[1].TimeDiff = FBCamera_0.Results.TimeDiff_ms;
			tmp = 1;
			i = 2;
		}
		else if (tmp){
			if (i < 20){
				BufferRes[i].X = FBCamera_0.Results.AxisX;
				BufferRes[i].Y = FBCamera_0.Results.AxisX;
				BufferRes[i].TimeDiff = FBCamera_0.Results.TimeDiff_ms;
				i++;
			}
		}
	}

	if ((GoalKeeper_0.isGoal1) || (GoalKeeper_0.isGoal2))
		tmp = 0;
	if (Reset){
		memset(&BufferRes,0,sizeof(BufferRes));
		i = 0;
		Reset = 0;
	}
}
```

#### Types.typ - Local data types
```iecst
TYPE
	LineChartAxis_type : 	STRUCT
		X : INT;
		Y : INT;
	END_STRUCT;
END_TYPE
```

- Visualisation Logical/mappView (not shown)

- Project.language (not shown)

### LibAsUDP1_ST.typ - Global data types
```iecst
(********************************************************************
 * COPYRIGHT -- Bernecker + Rainer
 ********************************************************************
 * File: Global.typ
 * Author: Bernecker + Rainer
 * Created: June 02, 2008
 ********************************************************************
 * Global data types of project LibAsUDP
 ********************************************************************)

TYPE
	LibAsUDP1_ST_typ : 	STRUCT  (*Datatyp for global Variables*)
		receive_data : STRING[500]; (*adress arguments*)
		send_data : STRING[500]; (*Data which should be sent*)
	END_STRUCT;
END_TYPE
```

### LibAsUDP1_ST.var - Global variables
```iecst
(********************************************************************
 * COPYRIGHT -- Bernecker + Rainer
 ********************************************************************
 * File: Global.var
 * Author: Bernecker + Rainer
 * Created: June 02, 2008
 ********************************************************************
 * Global variables of project LibAsUDP
 ********************************************************************)
VAR
	LibAsUDP1_ST : LibAsUDP1_ST_typ := (0); (*Data for AsUDP Global Variables*)
END_VAR
```

### Program Logical/Connection/Client (IEC) - AsUDP Client Application

#### Client.st - Cyclic code
```iecst
(********************************************************************
 * COPYRIGHT -- Bernecker + Rainer
 ********************************************************************
 * Program: Client
 * File: Client.st
 * Author: Bernecker + Rainer
 * Created: June 02, 2008
 ********************************************************************
 * Implementation of program Client
 ********************************************************************)

PROGRAM _CYCLIC

	hodnota := 10;

	CASE Client.sStep OF

		0:	(* Open UDP Port *)
			Client.UdpOpen_0.enable := 1;
			Client.UdpOpen_0.pIfAddr := 0;	(* Listen on all TCP/IP Interfaces*)
			Client.UdpOpen_0.port := port;	(* Port to listen*)
			Client.UdpOpen_0.options := 0;
			Client.UdpOpen_0;	(* Call the Function*)

			IF Client.UdpOpen_0.status = 0 THEN  (* UdpOpen successful*)
				Client.sStep := 1;
			ELSIF Client.UdpOpen_0.status = ERR_FUB_BUSY THEN  (* UdpOpen not finished -> redo *)
			  (* Busy *)
			ELSE  (* Goto Error Step *)
				Client.sStep := 10;
			END_IF

		1:	(* Send Data to the Server *)
			Client.server_address := adress;	(* IP Address of the Server *)
			Client.server_portnumber := port;	(* Port number of the Server *)

			memset(ADR(LibAsUDP1_ST.send_data),0,SIZEOF(LibAsUDP1_ST.send_data));

			strcpy(ADR(LibAsUDP1_ST.send_data),ADR(path));
			strcat(ADR(LibAsUDP1_ST.send_data),ADR(';'));
			strcat(ADR(LibAsUDP1_ST.send_data),ADR(arguments));

			Client.UdpSend_0.enable := 1;
			Client.UdpSend_0.ident := Client.UdpOpen_0.ident;	(* Connection Ident from AsUDP.UDP_Open *)
			Client.UdpSend_0.pHost := ADR(Client.server_address);
			Client.UdpSend_0.port := Client.server_portnumber;
			Client.UdpSend_0.pData := ADR(LibAsUDP1_ST.send_data);	(* Which data to send *)
			Client.UdpSend_0.datalen := SIZEOF(LibAsUDP1_ST.send_data);	(* Lenght of data to send *)
			Client.UdpSend_0.flags := 0;
			Client.UdpSend_0;	(* Call the Function*)

			IF Client.UdpSend_0.status = 0 THEN  (* Data sent *)
				Client.sStep := 2;
			ELSIF Client.UdpSend_0.status = ERR_FUB_BUSY THEN  (* UdpSend not finished -> redo *)
			  (* Busy *)
			ELSE  (* Goto Error Step *)
				Client.sStep := 10;
			END_IF

		2:	(* Receive Data from the Server *)
			Client.UdpRecv_0.enable := 1;
			Client.UdpRecv_0.ident := Client.UdpOpen_0.ident;  (* Connection Ident from AsUDP.UDP_Open *)
			Client.UdpRecv_0.pData	:= ADR(LibAsUDP1_ST.receive_data);  (* Where to store the incoming data *)
			Client.UdpRecv_0.datamax := SIZEOF(LibAsUDP1_ST.receive_data);  (* Lenght of data buffer *)
			Client.UdpRecv_0.flags := 0;
			Client.UdpRecv_0;  (* Call the Function*)

			IF Client.UdpRecv_0.status = 0 THEN  (* Data was received successfully -> Send next packet *)
				Client.sStep := 3;
				Client.no_data_received_count := 0;
			ELSIF Client.UdpRecv_0.status = udpERR_NO_DATA THEN  (* No data received - wait *)
			  (* No Data received *)
			  	Client.no_data_received_count := Client.no_data_received_count + 1;	(* Increase if no data are received *)
			ELSIF Client.UdpRecv_0.status = ERR_FUB_BUSY THEN  (* UdpRecv not finished -> redo *)
			  (* Busy *)
			ELSE  (* Goto Error Step *)
				Client.sStep := 10;
			END_IF

		3: (* Close connection *)
			Client.UdpClose_0.enable := 1;
			Client.UdpClose_0.ident := Client.UdpOpen_0.ident;  (* Connection Ident from AsUDP.UDP_Open *)
			Client.UdpClose_0;  (* Call the Function*)

			IF Client.UdpClose_0.status = 0 THEN  (* Close successful -> Reopen the interface *)
				Client.sStep := 10;
			ELSIF Client.UdpClose_0.status = ERR_FUB_BUSY THEN  (* UdpClose not finished -> redo *)
			  (* Busy *)
			ELSE  (* Goto Error Step *)
				Client.sStep := 10;
			END_IF

		10: (* Here some error Handling has to be implemented *)

	END_CASE

END_PROGRAM
```

#### Client.typ - UDP Client Variables
```iecst
(********************************************************************
 * COPYRIGHT -- Bernecker + Rainer
 ********************************************************************
 * Program: Client
 * File: Client.typ
 * Author: Bernecker + Rainer
 * Created: June 02, 2008
 ********************************************************************
 * Local data types of program Client
 ********************************************************************)

TYPE
	Client_typ : 	STRUCT  (*UDP Client Variables*)
		sStep : UINT := 10; (*UDP Client Step Variable*)
		server_address : STRING[20]; (*Address of the Server*)
		server_portnumber : UINT; (*Portnumber of the Server*)
		no_data_received_count : UINT; (*Counts up if no data are received*)
		UdpOpen_0 : UdpOpen; (*AsUDP.UdpOpen FUB*)
		UdpConnect_0 : UdpConnect; (*AsUDP.UdpConnect FUB*)
		UdpSend_0 : UdpSend; (*AsUDP.UdpSend FUB*)
		UdpRecv_0 : UdpRecv; (*AsUDP.UdpRecv FUB*)
		UdpDisconnect_0 : UdpDisconnect; (*AsUDP.UdpDisconnect FUB*)
		UdpClose_0 : UdpClose; (*AsUDP.UdpClose FUB*)
	END_STRUCT;
END_TYPE
```

#### Client.var - Data for Client Task
```iecst
(********************************************************************
 * COPYRIGHT -- Bernecker + Rainer
 ********************************************************************
 * Program: Client
 * File: Client.var
 * Author: Bernecker + Rainer
 * Created: June 02, 2008
 ********************************************************************
 * Local variables of program Client
 ********************************************************************)
VAR
	Client : Client_typ := (0); (*Data for Client Task*)
	hodnota : REAL;
END_VAR
```

Listed in the project but not available here: Logical/Global.typ, Logical/Libraries/IecCheck/IecCheck.fun, Logical/Libraries/IecCheck/IecCheck.st, Logical/Libraries/RO_Sensors/Constants.var, Logical/Libraries/RO_Sensors/Variables.var, Logical/Simulation/Technology/sim_cam_sens_sd_s/Types.typ, Logical/Simulation/Technology/sim_cam_sens_sd_s/Variables.var, Logical/Real_Game/Technology/cam_sens_sd_s/Variables.var
